FUNCTION_BLOCK ReedFlowMeter
VAR CONSTANT
	MAXLEN: UINT := 1000;
	TIMEUNITSPERSECOND: LINT := 10_000_000; // 100 ns per step
END_VAR
VAR
	fFrequencyToFlowScale: REAL := 0.28;
	fFlowRate: REAL;
	bReedSwitch AT %I*: BOOL;
	nIndex: UINT;
	timestamps: ARRAY [0..MAXLEN] OF ULINT;
	nTimeNow: ULINT; // 100 ns per unit
	nTriggerCount: UINT;
	nLoopIndex: UINT;
	trigger: R_TRIG;
END_VAR

// Koolance INS-FM19 flow meter
// simple reed contact switch
// frequency directly proportional to flow rate
// typical frequencies are <30 Hz, so no fast counter required

nTimeNow := F_GetSystemTime();
trigger(CLK:=bReedSwitch);
IF trigger.Q THEN
	timestamps[nIndex] := nTimeNow;
	nIndex := (nIndex + 1) MOD  MAXLEN;
END_IF

nTriggerCount := 0;
FOR nLoopIndex := 0 TO MAXLEN DO
	IF (ULINT_TO_LINT(nTimeNow) - ULINT_TO_LINT(timestamps[nLoopIndex])) < TIMEUNITSPERSECOND THEN
		nTriggerCount := nTriggerCount + 1;
	END_IF
END_FOR

fFlowRate := fFrequencyToFlowScale * nTriggerCount;

END_FUNCTION_BLOCK

(* stored: Version 1.1.0.1, ProductVersion 3.1.4024.12
   POU ReedFlowMeter: Id {b513db38-da5d-4cd1-bcee-622275ff067a}, SpecialFunc None *)
